FUNCTION_BLOCK Skill_Gripper_bistable_digout EXTENDS FB_1_Skill
VAR_INPUT
	Param : stParam_Gripper_bistable_digout;
	pTool: Pointer to FB_1_TOOL;
END_VAR
VAR_OUTPUT
END_VAR
VAR
	Phase: INT;
	tTimeout: TON;
END_VAR



IF rtStateChange.Q AND State = eState.Active THEN
	Phase := 10;
	ExecutionDone:=FALSE;
	ExecutionResult:=NONE;
	tTimeout(IN := FALSE);
END_IF

IF State <> eState.Active THEN
	Phase := 0;
	tTimeout(IN := FALSE);
END_IF

IF (Phase = 10) OR (Phase = 20) THEN
	IF pTool = 0 THEN
		ExecutionDone := TRUE;
		ExecutionResult := FAILURE;
		Messenger.AddError(eMessageCategories.MissingData,Path,'Gripper tool is not assigned');
		Phase := 0;
	ELSIF pTool^.pROB = 0 THEN
		ExecutionDone := TRUE;
		ExecutionResult := FAILURE;
		Messenger.AddError(eMessageCategories.MissingData,Path,'Gripper robot is not assigned');
		Phase := 0;
	END_IF
END_IF

IF Phase=10 THEN
	nCalledCmdID := pTool^.pROB^.SetDO(
		nOutput := Param.Pin,
		bValue := Param.ValueIfActiv);
	IF nCalledCmdID = 0 THEN
		ExecutionDone := TRUE;
		ExecutionResult := FAILURE;
		Messenger.AddWarn(eMessageCategories.ParentFailed,Path,'Robot rejected gripper command');
		Phase := 0;
	ELSE
		Phase := 20;
		tTimeout(IN := TRUE, PT := Param.TimeoutFailure);
	END_IF
END_IF


IF Phase=20 THEN
	tTimeout(IN := TRUE, PT := Param.TimeoutFailure);
	IF nCalledCmdID = pTool^.pROB^.CommandID THEN
		CASE pTool^.pROB^.CommandState OF
			INIT, ACKNOWLEDGE, RUNNING:
				Phase := 20;
			FINALIZED:
				ExecutionDone := TRUE;
				ExecutionResult := pTool^.pROB^.CommandResult;
				IF ExecutionResult <> SUCCESS THEN
					Messenger.AddWarn(eMessageCategories.ParentFailed,Path,'Gripper command failed');
				END_IF
				Phase := 0;
			ABORTED:
				ExecutionDone := TRUE;
				ExecutionResult := FAILURE;
				Messenger.AddWarn(eMessageCategories.ParentFailed,Path,'Gripper command aborted');
				Phase := 0;
		END_CASE
	END_IF

	IF (Phase = 20) AND tTimeout.Q THEN
		pTool^.pROB^.StopMotion();
		ExecutionDone := TRUE;
		ExecutionResult := FAILURE;
		Messenger.AddWarn(eMessageCategories.TimeoutFailure,Path,'Failed because timeout');
		Phase := 0;
	END_IF
END_IF

END_FUNCTION_BLOCK

(* stored: Version 1.1.0.1, ProductVersion 3.1.4026.18
   POU Skill_Gripper_bistable_digout: Id {a5a9cfad-4d81-4166-b0c8-d34649515f13}, SpecialFunc None *)
